# EPICS substitutions: example/exampleApp/Db/example.substitutions
#file E1214.template
#{
#pattern {P, R, PORT, IP_PORT}
#        {mkp:, E1214:, m1, m1ip}
#}

file E1241.template
{
pattern {P, R, PORT, IP_PORT}
        {mkp:, E1241:, m2, m2ip}
}

#file E1242.template
#{
#pattern {P, R, PORT, IP_PORT}
#        {mkp:, E1242:, m3, m3ip}
#}
